PROGRAM PRG_INJ
VAR
	i:INT;
	fullScale: REAL :=2000;
	DefaultSP :REAL:=0;
	rFULL_SCALE:REAL:=3000;//psig
END_VAR

// GCM
GCM_80(i_rFULL_SCALE := fullScale );
GFM_86(i_rFULL_SCALE:= rFULL_SCALE,rDefaultSP:=DefaultSP);

i:=i+1;
// Vent Valves
// interlock evaluation

VVC_80.i_xExtILK_OK := TRUE;//(NOT VVC_81.iq_stValve.q_xOPN_DO) AND(NOT VVC_82.iq_stValve.q_xOPN_DO); // Or we need to purge all the way up to the VCN
VVC_81.i_xExtILK_OK := (VVC_82.iq_stValve.q_xOPN_DO) AND (NOT VVC_83.iq_stValve.q_xOPN_DO) AND(NOT VVC_84.iq_stValve.q_xOPN_DO) AND (NOT VVC_85.iq_stValve.q_xOPN_DO) AND (NOT VVC_86.iq_stValve.q_xOPN_DO);// AND (NOT VVC_80.iq_stValve.q_xOPN_DO);
VVC_82.i_xExtILK_OK := (NOT VVC_83.iq_stValve.q_xOPN_DO) AND(NOT VVC_84.iq_stValve.q_xOPN_DO) AND (NOT VVC_85.iq_stValve.q_xOPN_DO) AND (NOT VVC_86.iq_stValve.q_xOPN_DO);// AND (NOT VVC_80.iq_stValve.q_xOPN_DO);

// instanitation
VVC_80(i_xExtILK_OK:= , i_xOverrideMode:= xOverrideMode, iq_stValve=> );
VVC_81(i_xExtILK_OK:= , i_xOverrideMode:= xOverrideMode, iq_stValve=> );
VVC_82(i_xExtILK_OK:= , i_xOverrideMode:= xOverrideMode, iq_stValve=> );



// Gas panel

// Interlock evaluation
VVC_83.i_xExtILK_OK := (NOT VVC_84.iq_stValve.q_xOPN_DO) AND (NOT VVC_85.iq_stValve.q_xOPN_DO) AND (NOT VVC_86.iq_stValve.q_xOPN_DO) AND (NOT VVC_81.iq_stValve.q_xOPN_DO) AND (NOT VVC_82.iq_stValve.q_xOPN_DO); // AND NOT bPurgeActive  
VVC_84.i_xExtILK_OK := (NOT VVC_83.iq_stValve.q_xOPN_DO) AND (NOT VVC_85.iq_stValve.q_xOPN_DO) AND (NOT VVC_86.iq_stValve.q_xOPN_DO) AND (NOT VVC_81.iq_stValve.q_xOPN_DO) AND (NOT VVC_82.iq_stValve.q_xOPN_DO); // AND NOT bPurgeActive  
VVC_85.i_xExtILK_OK := (NOT VVC_83.iq_stValve.q_xOPN_DO) AND (NOT VVC_84.iq_stValve.q_xOPN_DO) AND (NOT VVC_86.iq_stValve.q_xOPN_DO) AND (NOT VVC_81.iq_stValve.q_xOPN_DO) AND (NOT VVC_82.iq_stValve.q_xOPN_DO); // AND NOT bPurgeActive  
VVC_86.i_xExtILK_OK := (NOT VVC_83.iq_stValve.q_xOPN_DO) AND (NOT VVC_84.iq_stValve.q_xOPN_DO) AND (NOT VVC_85.iq_stValve.q_xOPN_DO) AND (NOT VVC_81.iq_stValve.q_xOPN_DO) AND (NOT VVC_82.iq_stValve.q_xOPN_DO);// AND NOT bPurgeActive 

//Gas Panel
VVC_83(i_xExtILK_OK:= , i_xOverrideMode:= xOverrideMode, iq_stValve=> );
VVC_84(i_xExtILK_OK:= , i_xOverrideMode:= xOverrideMode, iq_stValve=> );
VVC_85(i_xExtILK_OK:= , i_xOverrideMode:= xOverrideMode, iq_stValve=> );
VVC_86(i_xExtILK_OK:= , i_xOverrideMode:= xOverrideMode, iq_stValve=> );

RTD();

END_PROGRAM

(* stored: Version 1.1.0.1, ProductVersion 3.1.4022.18
   POU PRG_INJ: Id {4779f673-b478-4793-9f51-1eb8b319837c}, SpecialFunc None *)
